FUNCTION F_LogWarning : STRING;
VAR_INPUT
	Message : T_MaxString;
END_VAR

F_LogWarning := F_Logger(ADSLOG_MSGTYPE_WARN, Message);

END_FUNCTION

(* stored: Version 1.1.0.1, ProductVersion 3.1.4020.12
   POU F_LogWarning: Id {06f59f33-ec58-4ab0-babf-36fd7cd1be18}, SpecialFunc None *)
